RoboDK station: MoveBill.rdk

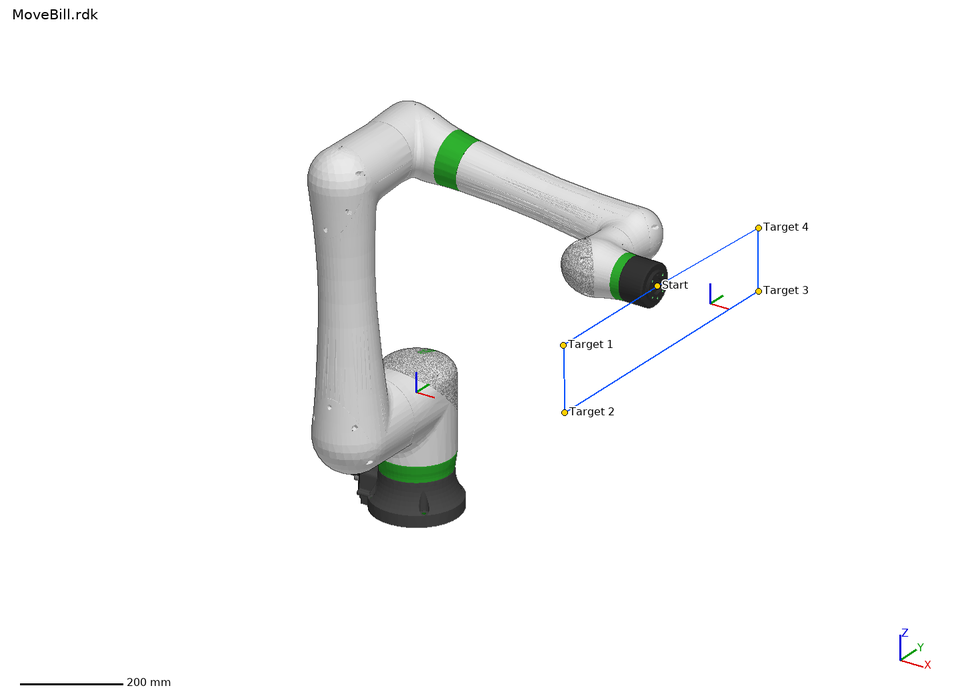
[picture v0: the station drawn from its stored meshes, robots at their saved joint values, targets as dots, program paths as lines]
Station MoveBill (saved by RoboDK 5.5.4). Poses are relative to the parent item; angles as X-Y-Z fixed-axis rotations.
Station parameters (name, value as stored): LIN64
  - frame Fanuc CRX-10iA Base at (0, 0, 245) mm
    - robot Fanuc CRX-10iA: 6 axes, payload 10 kg, reach 1249 mm, repeatability 0.05 mm, weight 40 kg
        modified DH rows (alpha deg, a mm, theta deg, d mm): 0, 0, 0, 245; -90, 0, -90, 0; 0, 540, 0, 0; -90, 0, 0, 540; 90, 0, 0, -150; -90, 0, 0, 160
        base shift (0, 0, -245) mm
        joint limits [-180, -180, -360, -190, -180, -190] to [180, 180, 430, 190, 180, 190]; home [0, 0, 0, 0, 0, 0]; saved at [0.211, -2.453, -6.216, -1.947, 6.219, 1.935]
  - frame Frame 2 at (800, -150, 720) mm
    - target Start (Cartesian target) at (-126.29, 1.98, 0.97) mm, rotated rx 0 ry -90 rz 180 deg; joints [0.211, -2.453, -6.216, -1.947, 6.219, 1.935] of Fanuc CRX-10iA
    - target Target 1 (Cartesian target) at (-126.29, -316.07, 0.97) mm, rotated rx 0 ry -90 rz 180 deg; joints [-37.318, 14.559, -19.122, 66.745, 41.288, -60.234] of Fanuc CRX-10iA
    - target Target 2 (Cartesian target) at (-126.29, -312.84, -145.61) mm, rotated rx 0 ry -90 rz 180 deg; joints [-34.395, 17.717, -31.944, 52.3, 45.556, -42.176] of Fanuc CRX-10iA
    - target Target 3 (Cartesian target) at (-126.29, 342.9, -145.61) mm, rotated rx 0 ry -90 rz 180 deg; joints [24.619, 3.092, -7.017, -75.072, 25.54, 73.539] of Fanuc CRX-10iA
    - target Target 4 (Cartesian target) at (-126.29, 342.9, -10.06) mm, rotated rx 0 ry -90 rz 180 deg; joints [14.17, -0.712, 6.488, -114.112, 15.557, 114.919] of Fanuc CRX-10iA
    - target Start (Cartesian target) at (-126.29, 1.98, 0.97) mm, rotated rx 0 ry -90 rz 180 deg; joints [0.211, -2.453, -6.216, -1.947, 6.219, 1.935] of Fanuc CRX-10iA
  - Python program testCRX10Model_10 (listed below)
  - Python program Prog2 (listed below)
  - program Prog3 (7 instructions, listed below)
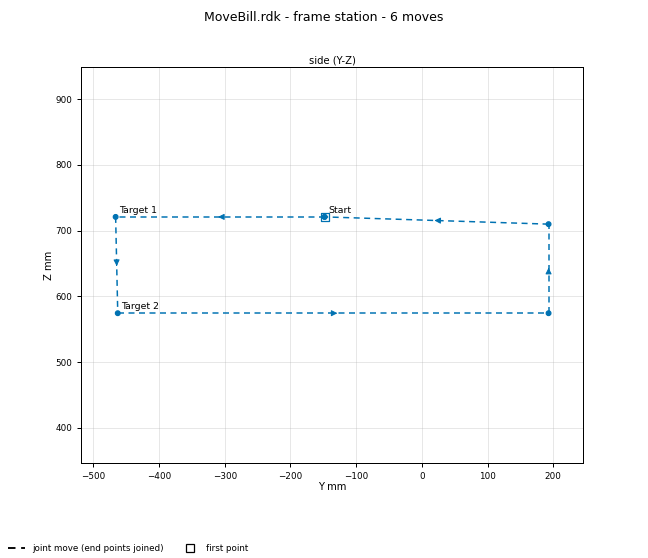
[picture p0: tool path of MoveBill.rdk in frame station, 6 of 6 moves have a stored position in this frame; points joined in program order, loops and branches not executed]

--- Python program testCRX10Model_10 ---
import time

from robodk.robolink import *                  # import the robolink library
RDK = Robolink()                        # connect to the RoboDK API (RoboDK starts if it has not started

robots = RDK.ItemList(ITEM_TYPE_ROBOT)
print(robots)


# tool  = RDK.Item('SCHUNK- 1321170 Co-act EGP-C 40-N-N-KTOE_ 0')                # Get an item named Tool (name in the RoboDK station tree)

robot = RDK.Item('', ITEM_TYPE_ROBOT)   # Get the first available robot


robot.Connect()
RDK.setRunMode(RUNMODE_RUN_ROBOT)
#RDK.setRunMode(RUNMODE_SIMULATE)
#frame = RDK.ItemUserPick('Select a reference frame', ITEM_TYPE_FRAME)   # Promt the user to select a reference frame
frame = RDK.Item('Frame 2', ITEM_TYPE_FRAME)

robot.setPoseFrame(frame)
# robot.setPoseTool(tool)

robot.setSpeed(speed_joints = 1000, speed_linear = 1000, accel_linear = 1000, accel_joints = 1000)

for i in range(0,5):
	print("Run: ", i)
	target = RDK.Item('Start', ITEM_TYPE_TARGET)   # Get a target called "turn1"
	robot.MoveJ(target)             # Move the robot to the target using the selected reference frame

	#time.sleep(1.0)

	target = RDK.Item('Target 1', ITEM_TYPE_TARGET)   # Get a target called "home"
	robot.MoveJ(target)             # Move the robot to the target using the selected reference frame

	target = RDK.Item('Target 2', ITEM_TYPE_TARGET)   # Get a target called "home"
	robot.MoveJ(target)             # Move the robot to the target using the selected reference frame

	target = RDK.Item('Target 3', ITEM_TYPE_TARGET)   # Get a target called "home"
	robot.MoveJ(target)             # Move the robot to the target using the selected reference frame

	target = RDK.Item('Target 4', ITEM_TYPE_TARGET)   # Get a target called "home"
	robot.MoveJ(target)             # Move the robot to the target using the selected reference frame

	target = RDK.Item('Start', ITEM_TYPE_TARGET)   # Get a target called "home"
	robot.MoveJ(target)             # Move the robot to the target using the selected reference frame

#	target = RDK.Item('Home', ITEM_TYPE_TARGET)   # Get a target called "home"
#	robot.MoveJ(target)             # Move the robot to the target using the selected reference frame

--- Python program Prog2 ---
# Type help("robodk.robolink") or help("robodk.robomath") for more information
# Press F5 to run the script
# Documentation: https://robodk.com/doc/en/RoboDK-API.html
# Reference:     https://robodk.com/doc/en/PythonAPI/robodk.html
# Note: It is not required to keep a copy of this file, your Python script is saved with your RDK project

# You can also use the new version of the API:
from robodk import robolink    # RoboDK API
from robodk import robomath    # Robot toolbox
RDK = robolink.Robolink()

# Forward and backwards compatible use of the RoboDK API:
# Remove these 2 lines to follow python programming guidelines
from robodk import *      # RoboDK API
from robolink import *    # Robot toolbox
# Link to RoboDK
# RDK = Robolink()

# Notify user:
print('To edit this program:\nright click on the Python program, then, select "Edit Python script"')

# Program example:
item = RDK.Item('base')
if item.Valid():
    print('Item selected: ' + item.Name())
    print('Item posistion: ' + repr(item.Pose()))

print('Items in the station:')
itemlist = RDK.ItemList()
print(itemlist)

# Provoking an exception will display the console output if you run this script from RoboDK
raise Exception('Program not edited.')

--- program Prog3 (robot Fanuc CRX-10iA) ---
  Set Ref.: Frame 2
  MoveJ (Start)
  MoveJ (Target 1)
  MoveJ (Target 2)
  MoveJ (Target 3)
  MoveJ (Target 4)
  MoveJ (Start)
